// TIA Portal V17 export
// export: Created 2025-03-05T08:03:36.4960693Z, ExportSetting WithDefaults, DisplayName Totally Integrated Automation Portal, DisplayVersion V17 Update 8, DisplayName TIA Portal Openness, DisplayVersion V17 Update 8, DisplayName TIA Portal Version Control Interface, DisplayVersion V17, DisplayName SINAMICS Startdrive Advanced, DisplayVersion V17 SP2, DisplayName SINAMICS Startdrive G110M, G120, G120C, G120D, G120P, G115D, DisplayVersion V17 SP2, DisplayName SINAMICS Startdrive G130, G150, S120, S150, SINAMICS MV, S210, DisplayVersion V17 SP2, DisplayName STEP 7 Professional, DisplayVersion V17 Update 8, DisplayName SINUMERIK ONE STEP 7 Toolbox, DisplayVersion V17 Update 12, DisplayName SINUMERIK 840D sl STEP 7 Toolbox, DisplayVersion V17 Update 12, DisplayName STEP 7 Safety, DisplayVersion V17 Update 6, DisplayName WinCC Advanced, DisplayVersion V17 Update 8
DATA_BLOCK "DB1022_PLC_CNC_DATA_SAFE"   // DB1022, F_DB
{ S7_Optimized_Access := 'TRUE'; DB_Accessible_From_OPC_UA := 'FALSE' }
VERSION : 0.1
// stored: AutoNumber false, DBAccessibleFromOPCUA false, DBAccessibleFromWebserver true
   VAR
      SEND_ERROR : Bool;
      SEND_SUBS_ON : Bool;
      RECEIVE_ERROR : Bool;   // COMMUNICATION ERROR
      RECEIVE_SUBS_ON : Bool;   // FAIL-SAFE VALUES ARE OUTPUT
      RECEIVE_ACK_REQ : Bool;   // ACKNOWLEDGMENT FOR REINTEGRATION OF SEND DATA REQUIRED
      RECEIVE_SENDMODE : Bool;   // F-CPU WITH SENDDP INSTRUCTION IS DISABLED SAFETY MODE
   END_VAR
BEGIN
END_DATA_BLOCK
